TYPE SwitchTable :
STRUCT
	
sName 	: STRING;
Signal	: BOOL;

END_STRUCT
END_TYPE

(* stored: Version 1.1.0.1, ProductVersion 3.1.4024.12
   DUT SwitchTable: Id {2976df91-dc83-4ecc-b1c2-f7bd7b9fc8fc} *)
